INTERFACE I_XP_Mover  EXTENDS I_CH_Object

METHOD AddToGroup : HRESULT
VAR_INPUT
	iGroup : I_XP_Group;
END_VAR
END_METHOD

{attribute 'monitoring':='call'}
PROPERTY CurrentTrack : I_XP_Track
GET
END_GET
END_PROPERTY

METHOD Disable : HRESULT
VAR_INPUT
END_VAR
END_METHOD

{attribute 'monitoring':='call'}
PROPERTY DistToParentStation : LREAL //Distance to the responsible parent station [mm]
GET
END_GET
END_PROPERTY

METHOD DistToTrack : LREAL
VAR_INPUT
	iTrack : I_XP_Track;
END_VAR
END_METHOD

METHOD Enable : HRESULT
VAR_INPUT
END_VAR
END_METHOD

{attribute 'OPC.UA.DA.Property' := '1'}
{attribute 'monitoring':='call'}
PROPERTY Feedback : I_XP_Feedback
GET
END_GET
END_PROPERTY

METHOD Halt : HRESULT
VAR_INPUT
END_VAR
END_METHOD

METHOD JoinTrack : HRESULT
VAR_INPUT
	iTrack : I_XP_Track;
END_VAR
END_METHOD

{attribute 'monitoring':='call'}
PROPERTY LastCmdTargedGap : LREAL
GET
END_GET
END_PROPERTY

{attribute 'monitoring':='call'}
PROPERTY LastCmdTargedPosition : LREAL
GET
END_GET
END_PROPERTY

{attribute 'monitoring':='call'}
PROPERTY LastCmdTargedTrack: I_XP_Track
GET
END_GET
END_PROPERTY

{attribute 'monitoring':='call'}
PROPERTY Mapped : BOOL //Project is mapped to MC (McToPlc and PlcToMc)
GET
END_GET
END_PROPERTY

{attribute 'monitoring':='call'}
PROPERTY Mode : MC_PLANAR_MOVER_COMMAND_MODE
GET
END_GET
END_PROPERTY

METHOD MoveA : HRESULT
VAR_INPUT
	fPosition : LREAL;
END_VAR
END_METHOD

METHOD MoveB : HRESULT
VAR_INPUT
	fPosition : LREAL;
END_VAR
END_METHOD

METHOD MoveC : HRESULT
VAR_INPUT
	fPosition : LREAL;
	
	(* Addition turns to move in modulo movement (positive or negative). *)
	additionalTurns : UDINT := 0;
	
	(* Direction in which the target is approached. *)
	direction : Tc3_Mc3Definitions.MC_DIRECTION := Tc3_Mc3Definitions.MC_DIRECTION.mcDirectionNonModulo;
END_VAR
END_METHOD

METHOD MoveOnTrack : HRESULT
VAR_INPUT
	ipTrack : I_XP_Track;
	fPosition : LREAL;
	fGap : LREAL;
END_VAR
END_METHOD

METHOD MoveOnTrack_ShortestWay : HRESULT
VAR_INPUT
	ipTrack : I_XP_Track;
	fPosition : LREAL;
	fGap : LREAL;
END_VAR
END_METHOD

METHOD MoveOnTrackToStation : HRESULT
VAR_INPUT
	ipStation : I_XP_Station;
	fGap : LREAL;
END_VAR
END_METHOD

{attribute 'monitoring':='call'}
(* Height that is used for internal collision checks.[mm] *)
PROPERTY MoverHeight : LREAL
GET
END_GET
END_PROPERTY

{attribute 'monitoring':='call'}
//Mover could not be detected or was removed from the system
PROPERTY MoverIsNotPresent : BOOL
GET
END_GET
END_PROPERTY

{attribute 'monitoring':='call'}
(* Width that is used for internal collision checks.[mm] *)
PROPERTY MoverWidth : LREAL
GET
END_GET
END_PROPERTY

METHOD MoveXY : HRESULT
VAR_INPUT
	fPosition_X : LREAL;
	fPosition_Y : LREAL;
END_VAR
END_METHOD

METHOD MoveZ : HRESULT
VAR_INPUT
	fPosition : LREAL;
END_VAR
END_METHOD

{attribute 'monitoring':='call'}
//Unique object ID
PROPERTY OID : OTCID
GET
END_GET
END_PROPERTY

{attribute 'monitoring':='call'}
PROPERTY ParentStation : I_XP_Station
GET
END_GET
SET
END_SET
END_PROPERTY

{attribute 'monitoring':='call'}
PROPERTY PlanarMover : REFERENCE TO MC_PlanarMover
GET
END_GET
END_PROPERTY

{attribute 'monitoring':='call'}
(* Provides the last valide planar mover setpoint XYZABC [mm] *)
PROPERTY PositionAtDisable : REFERENCE TO MoverVector
GET
END_GET
END_PROPERTY

{attribute 'monitoring':='call'}
PROPERTY PositionOnTrack : Lreal
GET
END_GET
END_PROPERTY

{attribute 'monitoring':='call'}
(* Provides the current planar mover setpoint XYZABC [mm] *)
PROPERTY PositionSet : REFERENCE TO MoverVector
GET
END_GET
END_PROPERTY

METHOD RemoveFromGroup : HRESULT
END_METHOD

METHOD Reset : HRESULT
VAR_INPUT
END_VAR
END_METHOD

{attribute 'monitoring':='call'}
PROPERTY Route : REFERENCE TO FB_CH_List
GET
END_GET
END_PROPERTY

{attribute 'monitoring':='call'}
(* Velocity is zero *)
PROPERTY Standstill : BOOL
GET
END_GET
END_PROPERTY

{attribute 'monitoring':='call'}
PROPERTY TargetStation : String
GET
END_GET
SET
END_SET
END_PROPERTY

PROPERTY TcIoXPlanarMover : Tc3_XPlanarUtility.I_TcIoXPlanarMover
GET
END_GET
END_PROPERTY

{attribute 'monitoring':='call'}
PROPERTY UtilityMover : Tc3_XPlanarUtility.I_McPlanarMover
GET
END_GET
END_PROPERTY

END_INTERFACE

(* stored: Version 1.1.0.1, ProductVersion 3.1.4024.12
   Itf I_XP_Mover: Id {567b42ec-b45f-4b7f-a752-c8a31c59e383}
   Folder Group: Id {98522917-210e-4a16-96b2-caa3ecaab952}
   Folder Movement: Id {45a88e98-b38f-4e20-a2fc-c8f2eacf66e9}
   Folder Power: Id {6ad90f0c-2e61-418b-aeeb-5501ac650e15}
   Folder Track: Id {72a1ce14-cdbe-4ed5-b425-caf348424991}
   Folder XPlanarUtility: Id {2df32512-d70c-4321-8df1-ac6cf839314b}
   Method AddToGroup: Id {73ea1ac0-7bcc-4b60-8e2d-1355b58a060f}
   Property CurrentTrack: Id {69c62c7e-fb39-45b5-890b-317f4f8b20cb}
   Get Get: Id {72537a94-dd35-48db-bd13-306cc94464af}
   Method Disable: Id {2706c01e-8eb0-4c7c-b9b9-bc6026ccda5a}
   Property DistToParentStation: Id {2c112004-530c-4dd4-a1ce-66f19e205f05}
   Get Get: Id {473b0278-14bf-4f75-8e75-ed9d5b853830}
   Method DistToTrack: Id {5cf89fed-3711-4b0d-8593-11510bed9c97}
   Method Enable: Id {654d96e4-cc81-417e-8487-9607e549968c}
   Property Feedback: Id {4b1f9a45-e49b-4af1-8aa6-8ecc374a291d}
   Get Get: Id {e2f4d9e9-82f0-4cee-b9a0-9923ba2b4974}
   Method Halt: Id {046b42e8-6abb-4fe8-9265-1f8f3f2517a1}
   Method JoinTrack: Id {31147787-1411-44ed-b2b6-87cbd46573b0}
   Property LastCmdTargedGap: Id {a496c8f2-826a-4cba-93fc-b9675765056e}
   Get Get: Id {c8f57789-8af3-4ab1-aa8e-508a9ec2bccc}
   Property LastCmdTargedPosition: Id {dee0ea17-c5b1-4e7e-a97c-14c2f5d3d740}
   Get Get: Id {be0d85eb-e04f-4493-ac36-6ef9ba5c8a87}
   Property LastCmdTargedTrack: Id {3feb4643-3533-4273-b62d-32158d27543a}
   Get Get: Id {86b72d7f-e015-4ccb-8a1d-8cbad564148e}
   Property Mapped: Id {29fba0cd-0241-4594-844a-64cae7f19898}
   Get Get: Id {e9c319e5-216e-440c-9fe6-3c8c426c4edc}
   Property Mode: Id {155121c8-381b-4cdd-941f-af7116491591}
   Get Get: Id {6de44ca8-561f-4669-bf03-9d7ea70002e0}
   Method MoveA: Id {b042fe17-0ef5-4fe5-b650-42edf05ed986}
   Method MoveB: Id {9231b9e0-0775-4a13-aa5e-9179ea891e32}
   Method MoveC: Id {2f4f8a50-5619-46a2-8f8d-5e794fe60f10}
   Method MoveOnTrack: Id {b8ed01ff-29a6-4dea-9a0a-82dda551f489}
   Method MoveOnTrack_ShortestWay: Id {9ef653d3-fa0c-469f-9110-14a92b28a19e}
   Method MoveOnTrackToStation: Id {e699b82c-ab17-485f-b20a-ce8928efd71e}
   Property MoverHeight: Id {76c6d44a-94ed-48c4-9cd2-c16943cbfbe2}
   Get Get: Id {f2df1a97-8161-4b33-9f5a-2f1a9f725c3c}
   Property MoverIsNotPresent: Id {e40a60ae-99d6-49fb-9646-536fda4eeb14}
   Get Get: Id {c2d50c85-1348-4406-b3e6-8ecfb2a1f6d9}
   Property MoverWidth: Id {42c814e0-a325-4307-ab17-9bd20fefdcf3}
   Get Get: Id {e1b9ed3e-d64e-4296-94c2-cbaaf162b575}
   Method MoveXY: Id {20f1e13d-5751-45ab-9270-b581d1f529c5}
   Method MoveZ: Id {06fa6a41-a0d9-4513-85f2-620cccb1c48f}
   Property OID: Id {35394ce9-108d-478b-a7be-1635eb9da0ae}
   Get Get: Id {002f69cf-fb5b-41bc-aab5-c98b0b8b64b5}
   Property ParentStation: Id {a0cc072f-0eb1-4b5e-912c-3e2bc5d0354b}
   Get Get: Id {9d350ef0-d0d0-4de4-b849-2ebb50e862c9}
   Set Set: Id {78b10601-2cc8-4447-941c-9745c3971f81}
   Property PlanarMover: Id {88fe9e0a-0e89-478c-b5f7-e56e3553bd03}
   Get Get: Id {525df7f7-9f93-49d6-a3f7-0c2b71648e31}
   Property PositionAtDisable: Id {c249cbc7-6194-4e84-afc7-5747aa64f16e}
   Get Get: Id {72308883-7511-4aff-bc17-cc1075676282}
   Property PositionOnTrack: Id {518cae7c-639f-4ece-a5ee-c588dfd0a161}
   Get Get: Id {c83c88c8-455b-4b56-a2c8-b018d056ed98}
   Property PositionSet: Id {fad00538-d046-475d-8f0f-0fc6a3c679d5}
   Get Get: Id {21971bf4-080a-478b-ae5f-8566ea986574}
   Method RemoveFromGroup: Id {cee4b8eb-11b5-4f44-b08a-00c260e6ab44}
   Method Reset: Id {52916818-fd48-4af4-99c7-22ba17a3ed7c}
   Property Route: Id {90767d52-dc47-4331-940e-058ec6f4c00c}
   Get Get: Id {e498b67f-8337-4325-997a-fa93ee597621}
   Property Standstill: Id {6b971fc0-1d52-4798-a038-7ace9a2ec219}
   Get Get: Id {b94c2963-6ded-418e-9184-4696eea57475}
   Property TargetStation: Id {97d05437-e2dc-4493-893c-aaa23f5d0855}
   Get Get: Id {26e06e6e-e8c2-43da-8d32-f6cc1563b105}
   Set Set: Id {e033f054-fad9-43c1-aff3-0a08f57a2cc8}
   Property TcIoXPlanarMover: Id {1c57778a-8bd4-481d-8c71-cc34d720286e}
   Get Get: Id {f5617ed4-9613-4bc1-a526-cb00742a4511}
   Property UtilityMover: Id {3ecc98c5-7410-414c-991b-689c7c0933df}
   Get Get: Id {5c891266-a2d4-4f64-9af6-dd01fffb81e0} *)
